Fanuc KAREL source: CA0106.KL

-- PROVISIONAL review KL for V1013-1; original PC SHA256 9beb93fc16c24716581ddcc09872696cfe51e12a9eac79cf1b2eb62a25da8161
-- Incomplete behavior may be omitted. Consult companion uncertainty JSON. Do not deploy.
PROGRAM CA0106
%NOLOCKGROUP
BEGIN
  -- UNRESOLVED_PC offsets 0-1; opcodes 7B
  -- UNRESOLVED_PC offsets 6-22; opcodes 2D,2E,69,7F
  -- UNRESOLVED_PC offsets 27-31; opcodes 7F
  -- UNRESOLVED_PC offsets 36-43; opcodes 9C,23
  -- UNRESOLVED_PC offsets 48-55; opcodes 9D,23
  -- UNRESOLVED_PC offsets 60-71; opcodes 2E,23
  -- UNRESOLVED_PC offsets 76-83; opcodes 9D,23
  -- UNRESOLVED_PC offsets 88-97; opcodes 3F,75
  -- UNRESOLVED_PC offsets 102-116; opcodes 2E,22,9D,33,35
  -- UNRESOLVED_PC offsets 121-135; opcodes 2E,22,9D,33,35
  -- UNRESOLVED_PC offsets 140-155; opcodes 2E,22,32,35
  -- UNRESOLVED_PC offsets 160-175; opcodes 2E,22,32,35
  -- UNRESOLVED_PC offsets 180-196; opcodes 27,22,AA,23
  -- UNRESOLVED_PC offsets 201-205; opcodes 7F
END CA0106
